FUNCTION_BLOCK AX_SPLIT (* Basic FB with empty ECC *)
  (* Standard: 61499-2; Description: Copyright (c) 2024 franz This program and the accompanying materials are made available under the terms of the Eclipse Public License 2.0 which is available at https://www.eclipse.org/legal/epl-2.0/ SPDX-License-Identifier: EPL-2.0 *)
  (* Version 1.0, 2024-10-24, franz *)
  PACKAGE io::adp;
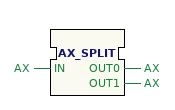
  SOCKETS
    IN : AX;
  END_SOCKETS
  PLUGS
    OUT0 : AX;
    OUT1 : AX;
  END_PLUGS
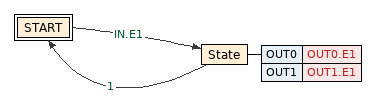
  EC_STATES
    START; (* Initial State *)
    State : OUT0 -> OUT0.E1, OUT1 -> OUT1.E1;
  END_STATES
  EC_TRANSITIONS
    State TO START := 1;
    START TO State := IN.E1;
  END_TRANSITIONS
  ALGORITHM OUT0 IN ST:
OUT0.D1 := IN.D1;
  END_ALGORITHM
  ALGORITHM OUT1 IN ST:
OUT1.D1 := IN.D1;
  END_ALGORITHM
END_FUNCTION_BLOCK
